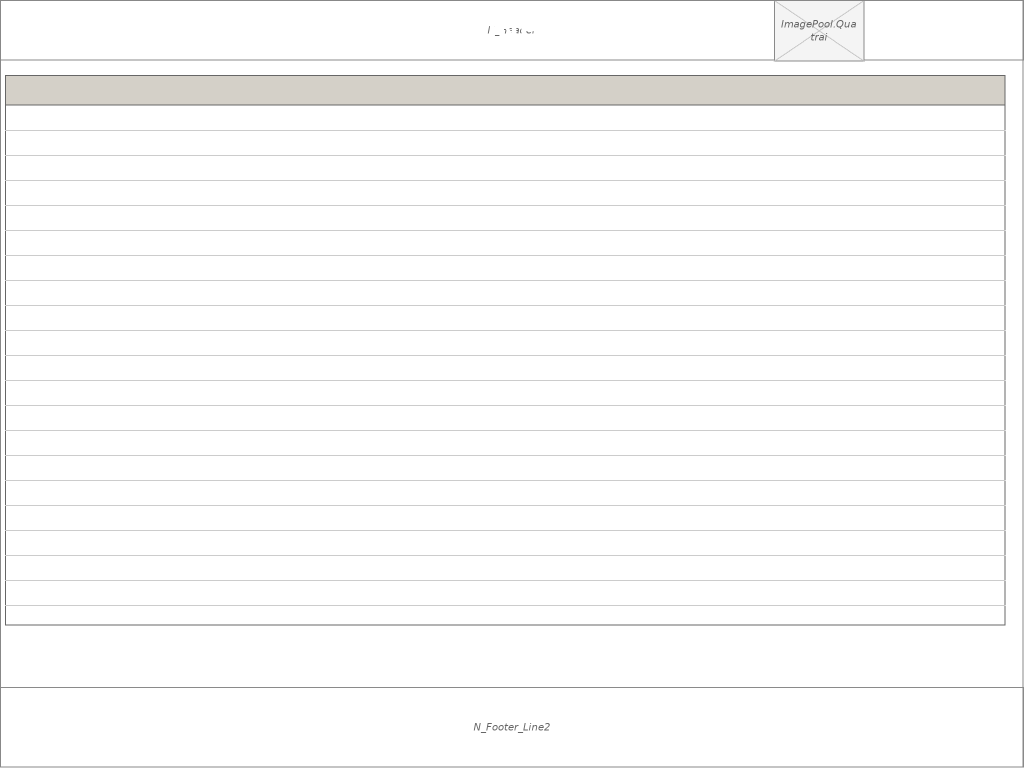
VISUALIZATION N_Alarm_1  // 1024x768
    Table (5,75 1000x550), invisible if: bVN, data array: AlarmList4
        p3854506369: AlarmList4[1,INDEX]
        p1892666644: AlarmList4[2,INDEX]
        p338671338: AlarmList[3,INDEX]
        p2170511999: AlarmList[4,INDEX]
        p511219082: Describe
        p1755163831: Status
        p4092479075: Time
        p1791247317: AlarmList4[3,INDEX]
        p262371475: AlarmList4[4,INDEX]
    Frame (0,687 1024x80)
        shows N_Footer_Line2()
    Frame (0,0 1024x60)
        shows N_Header()
    Textfield (353,5 400x50), "MÀN HÌNH LỖI TRẠM 2"
    Table (5,75 1000x550), invisible if: not bVN, data array: AlarmList2
        p3854506369: AlarmList2[1,INDEX]
        p1892666644: AlarmList2[2,INDEX]
        p338671338: AlarmList2[3,INDEX]
        p2170511999: AlarmList2[4,INDEX]
        p511219082: Mô tả
        p1755163831: Trạng thái
        p4092479075: Thời gian
    Image (774,0 90x61), image: ImagePool.Qua trai
        OnMouseClick: change screen: N_Alarm
END_VISUALIZATION

(* stored: Version 1.1.0.1, ProductVersion 3.1.4024.12
   Visu N_Alarm_1: Id {1a5f3dae-728e-4803-b05f-139364b63070} *)
